PROGRAM S_Etching
VAR_INPUT
	bInit				:BOOL:=FALSE;// 初始化状态 busy/done/errDone
	bTrig				:BOOL:=FALSE;// 执行触发 信号
	bReset				:BOOL:=FALSE;// 报错 复位
	bPause				:BOOL:=FALSE;// 暂停 运行
	bStop				:BOOL:=FALSE;// 停止 运行
	bAbort				:BOOL:=FALSE;// 中止 运行
	
END_VAR
VAR_OUTPUT
	busy				:BOOL;
	done				:BOOL;
	errDone				:BOOL;
END_VAR
VAR
	actStep				:ActStepBase;
END_VAR
VAR
	i: INT;
	t1:ton;
	t2:ton;
	t3:ton;
	notchoose:BOOL;
	timeOutTime:TIME:= T#120S;
	ventTime:TIME:=T#15S;
	safecheckTime:TIME:=T#2S;
	currentTimes:INT:=1;
	rfComControl:TON;
	rTrig:R_TRIG;
END_VAR

busy:=actStep.isBusy();
done:=actStep.isDone();
errDone:=actStep.isError();
actStep.Act_Pause(pause:=bPause);

IF bTrig THEN
	bTrig:=FALSE;
	IF NOT busy THEN
		actStep.Act_ex();
	END_IF
END_IF

//状态复位
IF bInit THEN
	bInit:=FALSE;
	Act_init_status();
END_IF

IF bAbort OR bStop THEN
	bAbort:=FALSE;
	bStop:=FALSE;
	Act_init_status();
	actStep.toZeroStep();
	S_CO_ControlRF.bStop:=TRUE;
	S_CO_ControlRF.bAbort:=TRUE;
	gRFComControl:=FALSE;
	gShowLogTextTitle:='NON';
END_IF
ActionRun(tempActStep:=actStep);
IF gRFComControl AND gICP.SourceRF.openRelay AND gICP.powerRF.openRelay THEN
	rfComControl(IN:=gICP.SourceRF.Get_Done_Open() AND gICP.PowerRF.Get_Done_Open(),PT:=UDINT_TO_TIME(gRFSetTime*1000));// 反射调整超时时间
	gRFRemainTime:=TIME_TO_UDINT(rfComControl.ET/1000);
	gRFRemainTime:=gRFSetTime-gRFRemainTime;
END_IF
rTrig(CLK:=gRFRemainTime=0);
IF rTrig.Q THEN
	gICP.SourceRF.Act_Close();
	gICP.PowerRF.Act_Close();
	gRFComControl:=FALSE;
END_IF

(*
---Trigger action
*)
METHOD Act_Ex : BOOL
VAR_INPUT
END_VAR
IF NOT busy THEN
	actStep.Act_ex();
	Act_Ex:=TRUE;
ELSE
	Act_Ex:=FALSE;
END_IF
END_METHOD

(*
---功能: 状态复位 busy/done/errDone;
*)
METHOD Act_Init_Status
VAR_INPUT
END_VAR
actStep.Act_Init();
END_METHOD

METHOD PRIVATE ActionRun
VAR_INPUT
	tempActStep:ITFActStep;
END_VAR
VAR_STAT//此处定义静态变量, 保证每次进入该函数时能够在线监控当前值
	tempStep:DINT;
END_VAR
tempStep:=tempActStep.getStep();
CASE tempStep OF
0:
	IF tempActStep.isEx() THEN
		tempActStep.setBusyFlag();
		tempActStep.toBeginStep();
	END_IF
	currentTimes:=1;
	t1(IN:= FALSE );
	t2(IN:= FALSE );
	t3(IN:= FALSE );
10:
	gShowLogTextTitle:='Etching';
	IF gRunningState<>RunningStatus.eErrorState THEN
		tempActStep.addStep(10,FALSE);
	ELSE
		error_Trigger(105);
	END_IF
	currentTimes:=1;
20:
	IF ControlMode.eSemiAutoMode=gCtrlMode OR ControlMode.eManualCtrMode=gCtrlMode THEN
		S_RoughPumping.Act_Init_Status();
		S_RoughPumping.Act_Ex();
		tempActStep.addStep(10,FALSE);
	ELSIF( ControlMode.eAutoCtrMode=gCtrlMode) THEN
		S_RoughPumping.Act_Init_Status();
		S_RoughPumping.Act_Ex();
		tempActStep.addStep(10,FALSE);
	ELSE
		tempActStep.toErrDoneStep();
	END_IF
30:
	IF S_RoughPumping.done THEN
		gShowLogTextTitle:='Etching';
		tempActStep.addStep(5,FALSE);
	END_IF
	IF S_RoughPumping.errDone THEN
		tempActStep.toErrDoneStep();
	END_IF	
35:
	tempActStep.addStep(5,TRUE);
40:
	IF gICP.HeMFC_SetFlowHMI<1 THEN
		tempActStep.toErrDoneStep();
		error_Trigger(200);
	ELSE
		tempActStep.addStep(10,FALSE);
	END_IF
50:// 记忆状态判断
	IF gWaferMemoryState=2 THEN
		gRunningLog.append(CONCAT('Etching POU Run:',DINT_TO_STRING(tempStep)));
		gRunningLog.append('Etching POU Run: wafer in chamber and etch done');
		tempActStep.toDoneStep();
	ELSIF gWaferMemoryState=1 THEN
		gRunningLog.append(CONCAT('Etching POU Run:',DINT_TO_STRING(tempStep)));
		gRunningLog.append('Etching POU Run: Wafer in chamber and no etch ');
		tempActStep.toStep(100,FALSE);// 直接进行Etch
	ELSIF gWaferMemoryState=0 THEN	
//		tempActStep.addStep(10,FALSE);// 先进行Load
		error_Trigger(116);
		tempActStep.toErrDoneStep();
	END_IF
100:
	tempActStep.addStep(10,TRUE);
110:
	tempActStep.addStep(10,FALSE);
120:
	IF NOT gICP.ForeLineGauge.error AND NOT gICP.LoadLockGauge.error AND NOT gICP.AIMGauge.error THEN
		tempActStep.addStep(10,FALSE);
	ELSE
		error_Trigger(107);
		tempActStep.toStep(10,FALSE);
	END_IF
130:
	IF gICP.ForlinLineValve.Act_Extend() AND gICP.PDV.Act_Open() THEN
		gRunningLog.append(CONCAT('Etching POU Run:',DINT_TO_STRING(tempStep)));
		gRunningLog.append('Etching POU Run: ForeLine Valve and PDV Open');
		tempActStep.addStep(10,FALSE);
	END_IF
140:
	IF (gICP.PDV.Get_Done_Ext() OR gICP.PDVOpenSensor) AND gICP.PDVOpenRelay AND gICP.ForlinLineValve.Get_Done_Ext() THEN
		gRunningLog.append(CONCAT('Etching POU Run:',DINT_TO_STRING(tempStep)));
		gRunningLog.append('Etching POU Run: ForeLine Valve and PDV Open Done');
		tempActStep.addStep(10,FALSE);
	END_IF
150:
	tempActStep.toStep(230,FALSE);	
230:
	tempActStep.addStep(10,TRUE);
240:	
	IF gICP.TruboPumNoRotation OR NOT(gICP.TruboPumAcc OR gICP.TruboPumDcc OR gICP.TruboPumNormal) AND FALSE THEN  //  临时屏蔽用
		IF gICP.TruboPum.Act_Open() THEN
			tempActStep.addStep(10,FALSE);
			gRunningLog.append(CONCAT('Etching POU Run:',DINT_TO_STRING(tempStep)));
			gRunningLog.append('Etching POU Run: TruboPum is not open');
		END_IF
	ELSE
		tempActStep.toStep(260,FALSE);
	END_IF
250:
	IF gICP.TruboPum.Get_Done_Open() AND gICP.TruboPumNormal AND gICP.TruboPumRotationSpeed>440 THEN
		gRunningLog.append(CONCAT('Etching POU Run:',DINT_TO_STRING(tempStep)));
		gRunningLog.append('Etching POU Run: TruboPum open Done');
		tempActStep.addStep(10,FALSE);
	END_IF
	IF  gICP.TruboPum.error THEN
		tempActStep.toErrDoneStep();
	END_IF
260:
	tempActStep.addStep(30,TRUE);//  临时屏蔽用
270:
	IF gICP.AIMValve.Act_Extend() THEN
		gRunningLog.append(CONCAT('Etching POU Run:',DINT_TO_STRING(tempStep)));
		gRunningLog.append('Etching POU Run:AIM Gauge open');
		tempActStep.addStep(10,FALSE);
	END_IF
280:
	t2(IN:= gICP.AIMGauge.outputValue<gUltimateVacuum AND gICP.AIMValve.Get_Done_Ext(),PT:=safecheckTime );
	IF t2.Q THEN
		t1(IN:= FALSE );
		t2(IN:= FALSE );
		t3(IN:= FALSE );
		gRunningLog.append(CONCAT('Etching POU Run:',DINT_TO_STRING(tempStep)));
		gRunningLog.append('Etching POU Run:AIM Gauge open Done and Preessure is Arrive');
		tempActStep.addStep(10,FALSE);
		RETURN;
	END_IF
	t3(IN:= TRUE,PT:=timeOutTime );
	IF t3.Q THEN
		t1(IN:= FALSE );
		t2(IN:= FALSE );
		t3(IN:= FALSE );
		error_Trigger(123);
		tempActStep.toErrDoneStep();
		RETURN;
	END_IF	
290:
	tempActStep.addStep(10,TRUE);
300:
	IF gICP.AIMValve.Act_Retract() THEN
		gRunningLog.append(CONCAT('Etching POU Run:',DINT_TO_STRING(tempStep)));
		gRunningLog.append('Etching POU Run:AIM Gauge Close');
		tempActStep.addStep(10,FALSE);
	END_IF
310:
	IF gICP.AIMValve.Get_Done_Ret() THEN
		gRunningLog.append(CONCAT('Etching POU Run:',DINT_TO_STRING(tempStep)));
		gRunningLog.append('Etching POU Run:AIM Gauge Close Done');
		tempActStep.addStep(10,FALSE);
	END_IF
320:
	tempActStep.addStep(10,TRUE);
330:
	IF gICP.LiftPinCyl.Act_Retract() THEN
		gRunningLog.append(CONCAT('Etching POU Run:',DINT_TO_STRING(tempStep)));
		gRunningLog.append('Etching POU Run:Lift PIN Down');
		tempActStep.addStep(10,FALSE);
	END_IF
340:
	IF gICP.LiftPinCyl.Get_Done_Ret() THEN
		tempActStep.addStep(10,FALSE);
	END_IF
350:
	tempActStep.addStep(10,TRUE);
360:
	IF gICP.ElectrodeCyl.Act_Extend() THEN
		gRunningLog.append(CONCAT('Etching POU Run:',DINT_TO_STRING(tempStep)));
		gRunningLog.append('Etching POU Run:ElectrodeCyl Up');
		tempActStep.addStep(10,FALSE);
	END_IF
370:
	IF gICP.ElectrodeCyl.Get_Done_Ext() THEN
		tempActStep.addStep(2,FALSE);
	END_IF
372:
	tempActStep.addStep(2,TRUE);
374:
	IF gICP.HeINValve.Act_Extend() THEN
		tempActStep.addStep(2,FALSE);
	END_IF
376:
	IF gICP.HeINValve.Get_Done_Ext() THEN
		tempActStep.addStep(2,FALSE);
	END_IF
378:
	tempActStep.addStep(2,FALSE);
380:
	tempActStep.addStep(10,TRUE);
390:
	IF currentTimes<=gShowNum THEN
		gICP.MFC1.setFlow:=STRING_TO_UDINT(gRecipeViewData[currentTimes].mfc1);
		gICP.MFC2.setFlow:=STRING_TO_UDINT(gRecipeViewData[currentTimes].mfc2);
		gICP.MFC3.setFlow:=STRING_TO_UDINT(gRecipeViewData[currentTimes].mfc3);
		gICP.MFC4.setFlow:=STRING_TO_UDINT(gRecipeViewData[currentTimes].mfc4);
		gICP.MFC5.setFlow:=STRING_TO_UDINT(gRecipeViewData[currentTimes].mfc5);
		gICP.MFC6.setFlow:=STRING_TO_UDINT(gRecipeViewData[currentTimes].mfc6);
		gICP.MFC7.setFlow:=STRING_TO_UDINT(gRecipeViewData[currentTimes].mfc7);
		gICP.MFC8.setFlow:=STRING_TO_UDINT(gRecipeViewData[currentTimes].mfc8);
		gICP.MFC9.setFlow:=STRING_TO_UDINT(gRecipeViewData[currentTimes].mfc9);
		tempActStep.addStep(10,FALSE);
		gRunningLog.append(CONCAT('Etching POU Run:',DINT_TO_STRING(tempStep)));
		gRunningLog.append('Etching POU Run:Set MFC Par');
		gRunningLog.append(CONCAT('Etching POU Run:',DINT_TO_STRING(tempStep)));
		gRunningLog.append(CONCAT('Etching POU Run:Current step is  ',INT_TO_STRING(currentTimes)));
	ELSE
		tempActStep.toStep(800,FALSE);////////////////////////////////////////////Done
	END_IF
	
400:
	IF gICP.S_GASBOX_AllMFCClearDoneStep THEN
		gICP.C_GASBOX_AllMFCSet:=TRUE;
		gICP.S_GASBOX_AllMFCSetDone:=FALSE;
		tempActStep.addStep(10,FALSE);
	END_IF
410:
	IF NOT gICP.C_GASBOX_AllMFCSet THEN
		tempActStep.addStep(10,FALSE);
	END_IF
420:
	IF gICP.S_GASBOX_AllMFCSetDone THEN
		gRunningLog.append(CONCAT('Etching POU Run:',DINT_TO_STRING(tempStep)));
		gRunningLog.append('Etching POU Run:Set MFC Par Done');
		tempActStep.addStep(10,FALSE);
	END_IF
430:
	tempActStep.addStep(10,TRUE);
440:
	gICP.C_GASBOX_AllGVAOpen:=TRUE;
	gRunningLog.append(CONCAT('Etching POU Run:',DINT_TO_STRING(tempStep)));
	gRunningLog.append('Etching POU Run:GAS Box GVA Open');
	tempActStep.addStep(10,FALSE);
450:
	IF gICP.S_GASBOX_AllGVAOpen THEN
		gRunningLog.append(CONCAT('Etching POU Run:',DINT_TO_STRING(tempStep)));
		gRunningLog.append('Etching POU Run:GAS Box GVA Open Done');
		tempActStep.addStep(10,FALSE);
	END_IF
460:
	t1(IN:=TRUE ,PT:=T#4S);
	IF t1.Q THEN
		t1(IN:= FALSE );
		t2(IN:= FALSE );
		t3(IN:= FALSE );
		tempActStep.addStep(10,FALSE);
	END_IF
470:
	IF gICP.S_GASBOX_AllMFCClearDone THEN// 全部MFC实际流量小于1
		tempActStep.addStep(10,FALSE);
		gRunningLog.append(CONCAT('Etching POU Run:',DINT_TO_STRING(tempStep)));
		gRunningLog.append('Etching POU Run:GAS Box GVB MFC flow is clear done');
	END_IF
480:
	tempActStep.addStep(10,TRUE);
490:
	gICP.C_GASBOX_AllGVBOpen:=TRUE;
	gRunningLog.append(CONCAT('Etching POU Run:',DINT_TO_STRING(tempStep)));
	gRunningLog.append('Etching POU Run:GAS Box GVB Open');
	tempActStep.addStep(10,FALSE);
500:
	IF gICP.S_GASBOX_AllGVBOpen THEN
		gRunningLog.append(CONCAT('Etching POU Run:',DINT_TO_STRING(tempStep)));
		gRunningLog.append('Etching POU Run:GAS Box GVB Open Done');
		tempActStep.addStep(10,FALSE);
	END_IF
510:	
	t1(IN:=TRUE ,PT:=T#4S);
	IF t1.Q THEN
		t1(IN:= FALSE );
		t2(IN:= FALSE );
		t3(IN:= FALSE );
		tempActStep.addStep(10,FALSE);
	END_IF
520:
	IF gICP.S_GASBOX_AllMFCSetEqual THEN
		gRunningLog.append(CONCAT('Etching POU Run:',DINT_TO_STRING(tempStep)));
		gRunningLog.append('Etching POU Run:GAS Box MFC Set Flow is arrive');
		tempActStep.addStep(10,FALSE);
	END_IF
530:
	tempActStep.addStep(10,TRUE);
540:
	IF gICP.ISOValve.Act_Extend() THEN
		gRunningLog.append(CONCAT('Etching POU Run:',DINT_TO_STRING(tempStep)));
		gRunningLog.append('Etching POU Run:ISO Valve Open');
		tempActStep.addStep(10,FALSE);
	END_IF
550:
	IF gICP.ISOValve.Get_Done_Ext() THEN
		tempActStep.addStep(10,FALSE);
	END_IF
560:
	tempActStep.addStep(10,TRUE);
570:
	gICP.PDV.Act_ChangePre(STRING_TO_REAL(gRecipeViewData[currentTimes].pdvPoint));
	gRunningLog.append(CONCAT('Etching POU Run:',DINT_TO_STRING(tempStep)));
	gRunningLog.append('Etching POU Run:PDV is change mode to preessur mode');
	tempActStep.addStep(10,FALSE);
580:
	IF gICP.PDV.Get_Done_Mode() THEN
		tempActStep.addStep(10,FALSE);
	END_IF
590:
	tempActStep.addStep(5,TRUE);
595:
	IF NOT gICP.S_MFCMonitFlowNotZero THEN
		tempActStep.addStep(5,FALSE);
	ELSE
		error_Trigger(120);
		tempActStep.toStep(590,FALSE);
		RETURN;
	END_IF
600:
	gRunningLog.append(CONCAT('Etching POU Run:',DINT_TO_STRING(tempStep)));
	gRunningLog.append('Etching POU Run:Set RF Par');
	gICP.SourceRF.HMIItf.setpower:=STRING_TO_UDINT(gRecipeViewData[currentTimes].rfPoint_Source);
	gICP.SourceRF.setpower:=gICP.SourceRF.HMIItf.setpower;
	gICP.SourceRF.Act_Write();
	tempActStep.addStep(10,FALSE);
610:
	IF gICP.SourceRF.HMIItf.setpower=gICP.SourceRF.setpower AND gICP.SourceRF.setpower=gICP.SourceRF.setpowerRead THEN
		tempActStep.addStep(10,FALSE);
	END_IF
620:
	gICP.PowerRF.HMIItf.setpower:=STRING_TO_UDINT(gRecipeViewData[currentTimes].rfPoint_Power);
	gICP.PowerRF.setpower:=gICP.PowerRF.HMIItf.setpower;
	gICP.PowerRF.Act_Write();
	gCO_ControlRFTime:=STRING_TO_UDINT(gRecipeViewData[currentTimes].etchTime);
	tempActStep.addStep(10,FALSE);
630:
	IF gICP.PowerRF.HMIItf.setpower=gICP.PowerRF.setpower AND gICP.PowerRF.setpower=gICP.PowerRF.setpowerRead THEN
		tempActStep.addStep(10,FALSE);
	END_IF
640:
	tempActStep.addStep(10,FALSE);
650:
	S_CO_ControlRF.Act_Init_Status();
	S_CO_ControlRF.Act_Ex();
	gRunningLog.append(CONCAT('Etching POU Run:',DINT_TO_STRING(tempStep)));
	gRunningLog.append('Etching POU Run:RF Open');
	tempActStep.addStep(5,FALSE);
655:
	IF S_CO_ControlRF.busy THEN
		tempActStep.addStep(5,FALSE);
	END_IF
660:
	IF S_CO_ControlRF.done THEN
		gRunningLog.append(CONCAT('Etching POU Run:',DINT_TO_STRING(tempStep)));
		gRunningLog.append('Etching POU Run:Etch Done');
		tempActStep.addStep(10,FALSE);
		RETURN;
	END_IF
	IF S_CO_ControlRF.errDone THEN
		gCO_ControlRFTimeRemain:=gCO_ControlRFTime;
		tempActStep.toStep(590,FALSE);
	END_IF	
665://  临时屏蔽用
	t1(IN:=TRUE ,PT:=T#10S);
	IF t1.Q THEN
		t1(IN:= FALSE );
		t2(IN:= FALSE );
		t3(IN:= FALSE );
		tempActStep.addStep(5,FALSE);
	END_IF
670:////////////////关气，关其他的东西，还原
	tempActStep.addStep(10,TRUE);
680:
	gICP.C_GASBOX_AllGVBClose:=TRUE;
	gRunningLog.append(CONCAT('Etching POU Run:',DINT_TO_STRING(tempStep)));
	gRunningLog.append('Etching POU Run:Gas Box GVB close');
	tempActStep.addStep(2,FALSE);
682:
	tempActStep.addStep(2,TRUE);
684:
	IF gICP.ForlinLineValve.Act_Extend() AND gICP.PDV.Act_Open() THEN
		gRunningLog.append(CONCAT('Etching POU Run:',DINT_TO_STRING(tempStep)));
		gRunningLog.append('Etching POU Run:PDV and ForeLine Open');
		tempActStep.addStep(2,FALSE);
	END_IF
686:
	IF gICP.ForlinLineValve.Get_Done_Ext() AND (gICP.PDV.Get_Done_Ext() OR gICP.PDVOpenSensor) THEN
//		gICP.PDV.Act_ChangePos();
		tempActStep.addStep(4,FALSE);
	END_IF
690:
	IF gICP.S_GASBOX_AllMFCClearDone THEN
		gRunningLog.append(CONCAT('Etching POU Run:',DINT_TO_STRING(tempStep)));
		gRunningLog.append('Etching POU Run:Gas Box flow is cleared done');
		tempActStep.addStep(10,FALSE);
	END_IF
700:
	t1(IN:=TRUE ,PT:=T#2S);
	IF t1.Q THEN
		t1(IN:= FALSE );
		t2(IN:= FALSE );
		t3(IN:= FALSE );
		tempActStep.addStep(10,FALSE);
	END_IF
710:
	tempActStep.addStep(10,TRUE);
720:
	gICP.C_GASBOX_AllMFCClear:=TRUE;
	gRunningLog.append(CONCAT('Etching POU Run:',DINT_TO_STRING(tempStep)));
	gRunningLog.append('Etching POU Run:Gas Box set flow is cleared');
	tempActStep.addStep(10,FALSE);
730:
	IF gICP.S_GASBOX_AllMFCClearDone THEN
		tempActStep.addStep(10,FALSE);
	END_IF
740:
	gICP.C_GASBOX_AllGVAClose:=TRUE;
	gRunningLog.append(CONCAT('Etching POU Run:',DINT_TO_STRING(tempStep)));
	gRunningLog.append('Etching POU Run:Gas Box GVA Close');
	tempActStep.addStep(10,FALSE);
750:
	t1(IN:=TRUE ,PT:=T#2S);
	IF t1.Q THEN
		t1(IN:= FALSE );
		t2(IN:= FALSE );
		t3(IN:= FALSE );
		tempActStep.addStep(10,FALSE);
	END_IF
760:
	tempActStep.addStep(10,TRUE);
770:
	tempActStep.addStep(10,FALSE);
780:
//	IF gICP.PDV.ReadState=XXX THEN // PDV 模式切换完成
//		tempActStep.addStep(10,FALSE);
//	END_IF
	tempActStep.addStep(10,FALSE);
790:
	tempActStep.toStep(380,FALSE);
	currentTimes:=currentTimes+1;
	gRunningLog.append(CONCAT('Etching POU Run:',DINT_TO_STRING(tempStep)));
	gRunningLog.append(CONCAT('The current number of steps plus 1 ',''));
800:
	tempActStep.addStep(5,FALSE);
805:
	tempActStep.addStep(2,TRUE);
807:
	IF gICP.HeINValve.Act_Retract() THEN
		tempActStep.addStep(3,FALSE);
	END_IF
810:
	IF gICP.HeINValve.Get_Done_Ret() THEN
		tempActStep.addStep(2,FALSE);
	END_IF
812:
	tempActStep.addStep(2,TRUE);
814:
	IF gICP.HePumValve.Act_Extend() THEN
		tempActStep.addStep(2,FALSE);
	END_IF
816:
	IF gICP.HePumValve.Get_Done_Ext() THEN
		tempActStep.addStep(1,FALSE);
	END_IF
817:
	t2(IN:=TRUE ,PT:=T#2S);
	IF t2.Q THEN
		t1(IN:= FALSE );
		t2(IN:= FALSE );
		t3(IN:= FALSE );
		tempActStep.addStep(1,FALSE);
	END_IF
818:
	t1(IN:=gICP.HeMFC_ActFlow<1 AND gICP.HeCheckGaugeReal<1 ,PT:=T#2S);
	IF t1.Q THEN
		t1(IN:= FALSE );
		t2(IN:= FALSE );
		t3(IN:= FALSE );
		gICP.HePumValve.Act_Retract();
		tempActStep.addStep(1,FALSE);
	END_IF
819:
	IF gICP.HePumValve.Get_Done_Ret() THEN
		tempActStep.addStep(1,FALSE);
	END_IF
820:
	IF gICP.ElectrodeCyl.Get_Done_Ret() THEN
		tempActStep.addStep(20,FALSE);
	ELSE
		IF gICP.ElectrodeCyl.Act_Retract() THEN
			tempActStep.addStep(10,FALSE);
		END_IF
	END_IF
830:
	IF gICP.ElectrodeCyl.Get_Done_Ret() THEN
		tempActStep.addStep(10,FALSE);
	END_IF
840:
	IF gICP.LiftPinCyl.Get_Done_Ret() THEN
		tempActStep.addStep(20,FALSE);
	ELSE
		IF gICP.LiftPinCyl.Act_Retract() THEN
			tempActStep.addStep(10,FALSE);
		END_IF
	END_IF
850:
	IF gICP.LiftPinCyl.Get_Done_Ret() THEN
		tempActStep.addStep(10,FALSE);
	END_IF
860:
	tempActStep.toStep(1000,FALSE);
1000:
	tempActStep.toDoneStep();

60000://Done
	tempActStep.setDoneFlag();
	tempActStep.toZeroStep();
	gWaferMemoryState:=2;
	ups_CX51X0.Act_Wrtie();
	gRunningLog.append('Etching POU Run:----Finish----');
	gRFComControl:=FALSE;
65000://Error
	tempActStep.setErrDoneFlag();
	tempActStep.toZeroStep();
	gRFComControl:=FALSE;
END_CASE
END_METHOD

END_PROGRAM

(* stored: Version 1.1.0.1, ProductVersion 3.1.4024.12
   POU S_Etching: Id {b6c2180f-56dc-49d8-a717-40b6200f35a3}, SpecialFunc None
   Folder Private: Id {5fc2896d-8763-4e02-983c-2edb2f09ad3f}
   Method Act_Ex: Id {9231d7ef-7988-4eb2-bc4c-1c8b40de6b16}
   Method Act_Init_Status: Id {4fc5e96c-6afd-4f7d-9bcf-b8a9cf1d5586}
   Method ActionRun: Id {b7cebe4e-80e4-4a3d-bf6b-1b34b2138e9a} *)
